FUNCTION_BLOCK MCCPower (* Composite Function Block Type *)
  (* Standard: 61499-2 *)
  (* Version 0.0, 3/8/2024, SESA371406, Schneider Electric, template *)
  PACKAGE SE.Nereda;
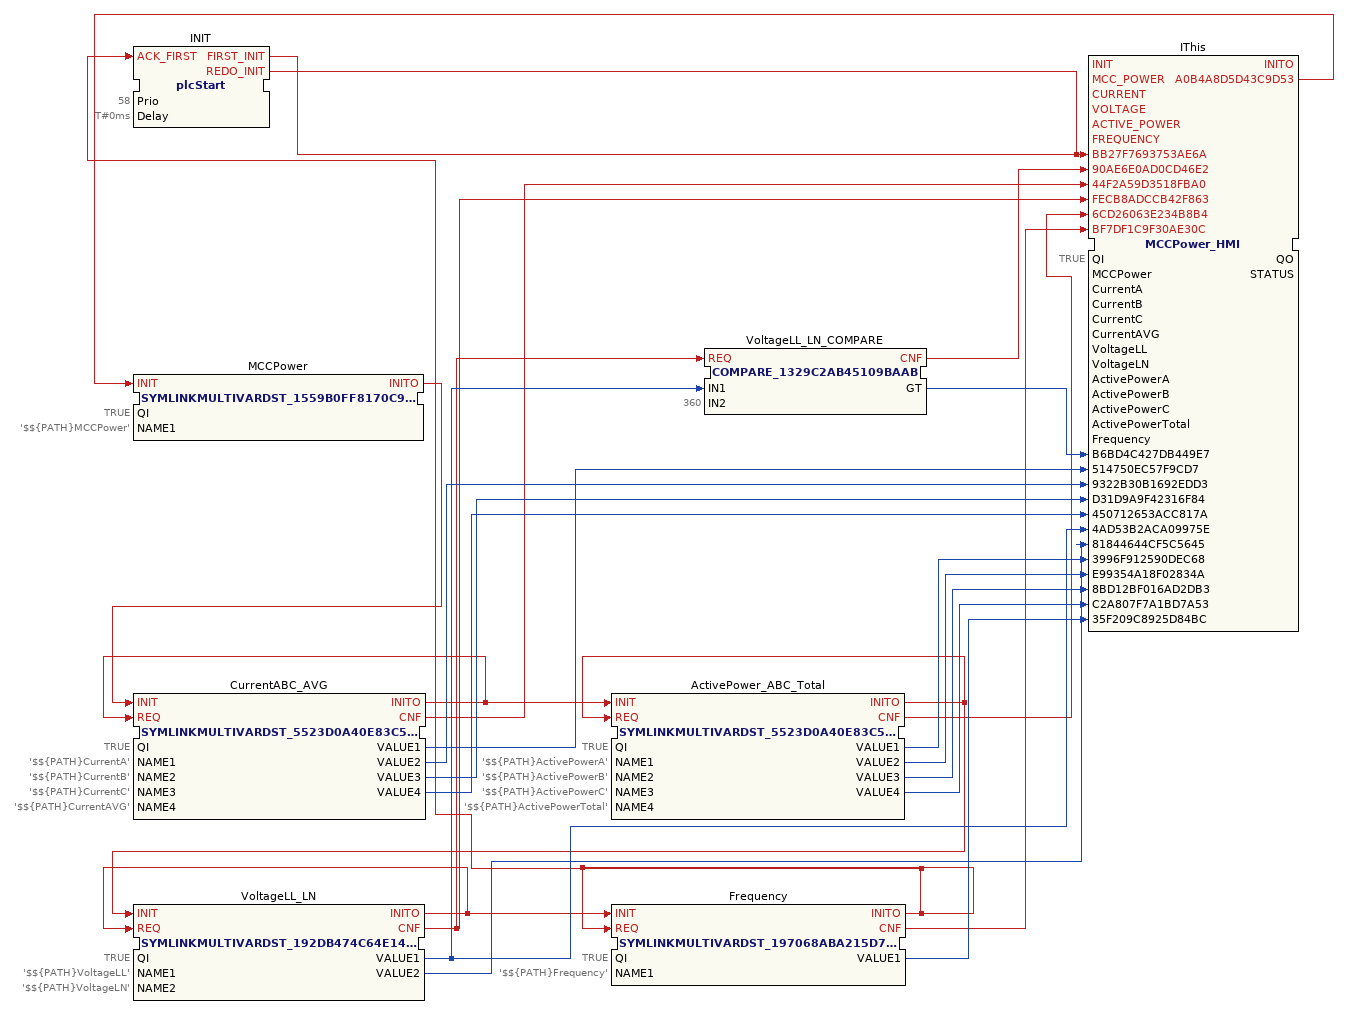
  FBS
    IThis : MCCPower_HMI(QI := TRUE);
    MCCPower : SYMLINKMULTIVARDST_1559B0FF8170C9BA0(QI := TRUE, NAME1 := '$${PATH}MCCPower'); {SET_ATTRIBUTE(Configuration.GenericFBType.InterfaceParams, Runtime.System#I:=1;VALUE${I$}:BOOL)}
    CurrentABC_AVG : SYMLINKMULTIVARDST_5523D0A40E83C5C4(QI := TRUE, NAME1 := '$${PATH}CurrentA', NAME2 := '$${PATH}CurrentB', NAME3 := '$${PATH}CurrentC', NAME4 := '$${PATH}CurrentAVG'); {SET_ATTRIBUTE(Configuration.GenericFBType.InterfaceParams, Runtime.System#I:=4;VALUE${I$}:REAL,REAL,REAL,REAL)}
    VoltageLL_LN : SYMLINKMULTIVARDST_192DB474C64E14111(QI := TRUE, NAME1 := '$${PATH}VoltageLL', NAME2 := '$${PATH}VoltageLN'); {SET_ATTRIBUTE(Configuration.GenericFBType.InterfaceParams, Runtime.System#I:=2;VALUE${I$}:REAL,REAL)}
    ActivePower_ABC_Total : SYMLINKMULTIVARDST_5523D0A40E83C5C4(QI := TRUE, NAME1 := '$${PATH}ActivePowerA', NAME2 := '$${PATH}ActivePowerB', NAME3 := '$${PATH}ActivePowerC', NAME4 := '$${PATH}ActivePowerTotal'); {SET_ATTRIBUTE(Configuration.GenericFBType.InterfaceParams, Runtime.System#I:=4;VALUE${I$}:REAL,REAL,REAL,REAL)}
    Frequency : SYMLINKMULTIVARDST_197068ABA215D7EBA(QI := TRUE, NAME1 := '$${PATH}Frequency'); {SET_ATTRIBUTE(Configuration.GenericFBType.InterfaceParams, Runtime.System#I:=1;VALUE${I$}:REAL)}
    VoltageLL_LN_COMPARE : COMPARE_1329C2AB45109BAAB(IN2 := 360); {SET_ATTRIBUTE(Configuration.GenericFBType.InterfaceParams, Runtime.Standard#CNT:=2;IN${CNT$}:REAL)}
    INIT : plcStart(Prio := 58, Delay := T#0ms);
  END_FBS
  EVENT_CONNECTIONS
    MCCPower.INITO TO CurrentABC_AVG.INIT;
    CurrentABC_AVG.INITO TO ActivePower_ABC_Total.INIT;
    ActivePower_ABC_Total.INITO TO VoltageLL_LN.INIT;
    VoltageLL_LN.INITO TO Frequency.INIT;
    Frequency.INITO TO INIT.ACK_FIRST;
    CurrentABC_AVG.INITO TO CurrentABC_AVG.REQ;
    ActivePower_ABC_Total.INITO TO ActivePower_ABC_Total.REQ;
    Frequency.INITO TO Frequency.REQ;
    VoltageLL_LN.INITO TO VoltageLL_LN.REQ;
    VoltageLL_LN.CNF TO VoltageLL_LN_COMPARE.REQ;
    INIT.FIRST_INIT TO IThis.BB27F7693753AE6A;
    VoltageLL_LN_COMPARE.CNF TO IThis.90AE6E0AD0CD46E2;
    CurrentABC_AVG.CNF TO IThis.44F2A59D3518FBA0;
    VoltageLL_LN.CNF TO IThis.FECB8ADCCB42F863;
    ActivePower_ABC_Total.CNF TO IThis.6CD26063E234B8B4;
    Frequency.CNF TO IThis.BF7DF1C9F30AE30C;
    IThis.A0B4A8D5D43C9D53 TO MCCPower.INIT;
    INIT.REDO_INIT TO IThis.BB27F7693753AE6A;
  END_CONNECTIONS
  DATA_CONNECTIONS
    VoltageLL_LN.VALUE1 TO VoltageLL_LN_COMPARE.IN1;
    VoltageLL_LN_COMPARE.GT TO IThis.B6BD4C427DB449E7;
    CurrentABC_AVG.VALUE1 TO IThis.514750EC57F9CD7;
    CurrentABC_AVG.VALUE2 TO IThis.9322B30B1692EDD3;
    CurrentABC_AVG.VALUE3 TO IThis.D31D9A9F42316F84;
    CurrentABC_AVG.VALUE4 TO IThis.450712653ACC817A;
    VoltageLL_LN.VALUE1 TO IThis.4AD53B2ACA09975E;
    VoltageLL_LN.VALUE2 TO IThis.81844644CF5C5645;
    ActivePower_ABC_Total.VALUE1 TO IThis.3996F912590DEC68;
    ActivePower_ABC_Total.VALUE2 TO IThis.E99354A18F02834A;
    ActivePower_ABC_Total.VALUE3 TO IThis.8BD12BF016AD2DB3;
    ActivePower_ABC_Total.VALUE4 TO IThis.C2A807F7A1BD7A53;
    Frequency.VALUE1 TO IThis.35F209C8925D84BC;
  END_CONNECTIONS
END_FUNCTION_BLOCK
